FUNCTION_BLOCK UnitTestPrinter
VAR_INPUT
END_VAR
VAR_OUTPUT
END_VAR
VAR
    messageBuilder: SimpleStringBuilder;
END_VAR

METHOD getFailureMessage : MaxString
VAR_INPUT
    expected: ANY;
    actual: ANY;
    message: MaxString;
    path: MaxString;
END_VAR
VAR
    messageToAppend: MaxString;
END_VAR
messageToAppend := 'FAILED TEST $'';
messageBuilder.append(messageToAppend);
messageBuilder.append(path);
messageToAppend := '$', EXP: ';
messageBuilder.append(messageToAppend);
messageBuilder.append(expected);
messageToAppend := ', ACT: ';
messageBuilder.append(messageToAppend);
messageBuilder.append(actual);
messageToAppend := ', MSG: ';
messageBuilder.append(messageToAppend);
messageBuilder.append(message);

getFailureMessage := messageBuilder.toString();
END_METHOD

METHOD printFailure
VAR_INPUT
    expected: MaxString;
    actual: MaxString;
    message: MaxString;
    path: MaxString;
END_VAR
VAR
    failureMessage: MaxString;
END_VAR
failureMessage := getFailureMessage(expected, actual, message, path);
END_METHOD

END_FUNCTION_BLOCK

(* stored: Version 1.1.0.1, ProductVersion 3.1.4022.12
   POU UnitTestPrinter: Id {c8b5c401-57cf-4e84-8c94-4746649c8d15}, SpecialFunc None
   Method getFailureMessage: Id {9dc6d79a-5505-4a87-87c3-d856af6043df}
   Method printFailure: Id {af4e89be-6949-40ab-9696-5dfe4e50e8cf} *)
